TYPE ST185_Recipe_t : 
STRUCT
    xUseVerLeft  : BOOL; // Is the left vertical picker element is used
    xUseVerRight : BOOL; // Is the right vertical picker element is used
END_STRUCT
END_TYPE

(* stored: Version 1.1.0.1, ProductVersion 3.1.4024.6
   DUT ST185_Recipe_t: Id {33785acb-0897-480e-937a-e0929462af23} *)
